// TIA Portal V17 export
// export: Created 2023-05-07T12:12:09.3609887Z, ExportSetting WithDefaults, DisplayName Totally Integrated Automation Portal, DisplayVersion V17, DisplayName TIA Portal Openness, DisplayVersion V17, DisplayName TIA Portal Version Control Interface, DisplayVersion V17, DisplayName TIA Portal Test Suite Advanced, DisplayVersion V17, DisplayName STEP 7 Professional, DisplayVersion V17, DisplayName SIMATIC Energy Suite, DisplayVersion V17, DisplayName STEP 7 Safety, DisplayVersion V17, DisplayName WinCC Professional, DisplayVersion V17
FUNCTION_BLOCK "StartStop"   // FB11, LAD
TITLE = StartStop
{ S7_Optimized_Access := 'TRUE' }
VERSION : 0.1
// stored: AutoNumber true, IsIECCheckEnabled false, IsRetainMemResEnabled false, MemoryReserve 100, SetENOAutomatically false, UDAEnableTagReadback false
   VAR_INPUT
      Start : Bool;
      Stop : Bool;
   END_VAR
   VAR_OUTPUT
      Q : Bool;
   END_VAR
   VAR
      statSR : Bool;
      statRisEdge : Bool;
   END_VAR
   VAR_TEMP   // added for the SCL form of the ladder/FBD networks
      _w1 : Bool;
   END_VAR
BEGIN

REGION Network 1: P_Trig && SR
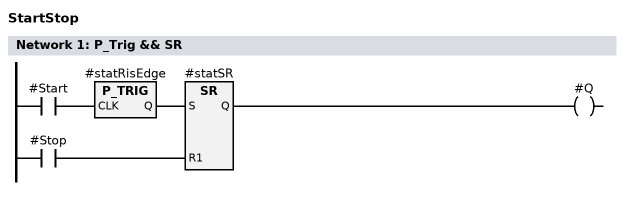
   RUNG wire#powerrail
      Contact( #Start )
      P_Trig( #statRisEdge )
      S_SR(operand := #statSR, r1 := wire#w1)
      Coil( #Q )
   END_RUNG
   RUNG wire#powerrail
      Contact( #Stop )
   END_RUNG wire#w1
   // the same network as SCL:
   #_w1 := #Start AND NOT #statRisEdge;   // rising edge
   #statRisEdge := #Start;
   IF #_w1 THEN
       #statSR := TRUE;   // SR flip-flop
   END_IF;
   IF #Stop THEN #statSR := FALSE; END_IF;
   #Q := #statSR;
END_REGION
END_FUNCTION_BLOCK
